// TIA Portal V20 export
// export: Created 2025-09-12T17:59:00.0000000Z, ExportSetting WithDefaults
FUNCTION_BLOCK "FB400_EM_Damper"   // FB, SCL
TITLE = EM-400: Damper Control
AUTHOR : Dallas Levine
VERSION : 0.1
// This block contains all logic for the Damper Equipment Module (EM-400).
// stored: AutoNumber true, IsRetain false
   VAR_INPUT
      Enable : Bool;   // Enables the block's execution.
   END_VAR
   VAR
      UDT : "UDT400_EM_Damper";   // The data interface for the Damper Equipment Module.
      Feedback_Fault_Timer : TON_TIME;   // Timer for the feedback fault delay.
   END_VAR
   VAR CONSTANT
      FEEDBACK_TOLERANCE : Real := 10.0;   // Allowable deviation between command and feedback (%).
      FEEDBACK_DELAY : Time := T#60s;   // Time delay before a feedback mismatch becomes an alarm.
   END_VAR
BEGIN
   REGION Main Logic 
   IF #Enable THEN
    (/**/) #Feedback_Fault_Timer(IN:= ABS(FV:=#UDT.Damper_Pos_Cmd_AO - #UDT.Damper_Pos_Fdbk_AI) > #FEEDBACK_TOLERANCE,
           PT:= #FEEDBACK_DELAY);
    #UDT.Damper_Failure_Alm := #Feedback_Fault_Timer.Q;
   ELSE
    (/**/) #UDT.Damper_Failure_Alm := FALSE;
   END_IF;
   END_REGION
END_FUNCTION_BLOCK
